TYPE ST_MessageBoxText :
STRUCT
	
	sText	: STRING;
	nColor	: DWORD;	

END_STRUCT
END_TYPE

(* stored: Version 1.1.0.1, ProductVersion 3.1.4024.13
   DUT ST_MessageBoxText: Id {29138eaa-499a-4e30-ae55-308b9de90680} *)
